PROGRAM VisionJog
VAR
	State:INT;
	
END_VAR

IF GVL.Mode = Modes.MAN THEN
	GVL.Vision.SingleShot(Enable:=HMI.Bt_ActivateSingle, 
						Execute:=HMI.Bt_Shot,
						Q=>GVL.VisionResults,
						Measurement=>HMI.L_NewMeasurement);
    GVL.Vision.ContinuousShot(Enable:=HMI.Bt_ActivateContinuous,
						Q=>GVL.VisionResults);
ELSE
	HMI.Bt_ActivateSingle:=FALSE;
	HMI.Bt_ActivateContinuous:=FALSE;
END_IF

END_PROGRAM

(* stored: Version 1.1.0.1, ProductVersion 3.1.4024.9
   POU VisionJog: Id {1712aba2-8ad2-43ea-86d8-883fbfc4e967}, SpecialFunc None *)
